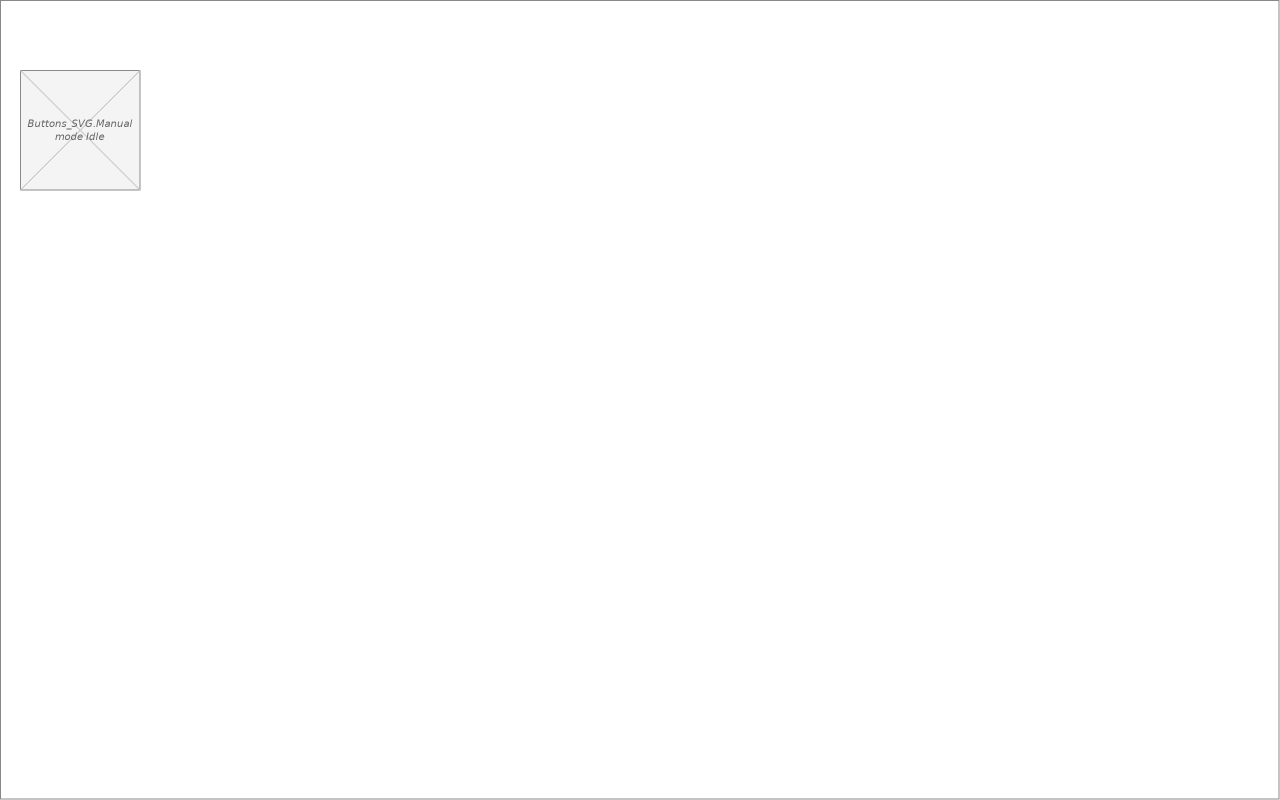
VISUALIZATION toManualButton  // 1280x800
    Image (20,70 120x120), image: Buttons_SVG.Manual mode Idle
        OnMouseClick: toggle GVL_HMI.bCmdManual
END_VISUALIZATION

(* stored: Version 1.1.0.1, ProductVersion 3.1.4024.10
   Visu toManualButton: Id {e5e337c4-6df6-4290-a08c-2b3898e12bd3} *)
